// TIA Portal V17 export
// export: Created 2025-03-13T10:29:45.3472643Z, ExportSetting WithDefaults, DisplayName Totally Integrated Automation Portal, DisplayVersion V17 Update 8, DisplayName TIA Portal Openness, DisplayVersion V17 Update 8, DisplayName TIA Portal Version Control Interface, DisplayVersion V17, DisplayName SINAMICS Startdrive Advanced, DisplayVersion V17 SP2, DisplayName SINAMICS Startdrive G110M, G120, G120C, G120D, G120P, G115D, DisplayVersion V17 SP2, DisplayName SINAMICS Startdrive G130, G150, S120, S150, SINAMICS MV, S210, DisplayVersion V17 SP2, DisplayName STEP 7 Professional, DisplayVersion V17 Update 8, DisplayName SINUMERIK ONE STEP 7 Toolbox, DisplayVersion V17 Update 12, DisplayName SINUMERIK 840D sl STEP 7 Toolbox, DisplayVersion V17 Update 12, DisplayName STEP 7 Safety, DisplayVersion V17 Update 6, DisplayName WinCC Advanced, DisplayVersion V17 Update 8
FUNCTION "FC4020_PART_PRESENT_CONTROL_U02_STA_1" : Void   // FC4020, LAD
{ S7_Optimized_Access := 'TRUE' }
VERSION : 0.1
// stored: AutoNumber false, IsIECCheckEnabled false, SetENOAutomatically false, UDAEnableTagReadback false
   VAR_TEMP
      SENSOR_VALUE_AUX : Real;
      DIV_AUX : Real;
      RESULT_AUX : Real;
      TOTAL_AUX : Real;
      SUP_LIM : Real;
      INF_LIM : Real;
   END_VAR
BEGIN

REGION Network 1: PART PRESENT INPUT
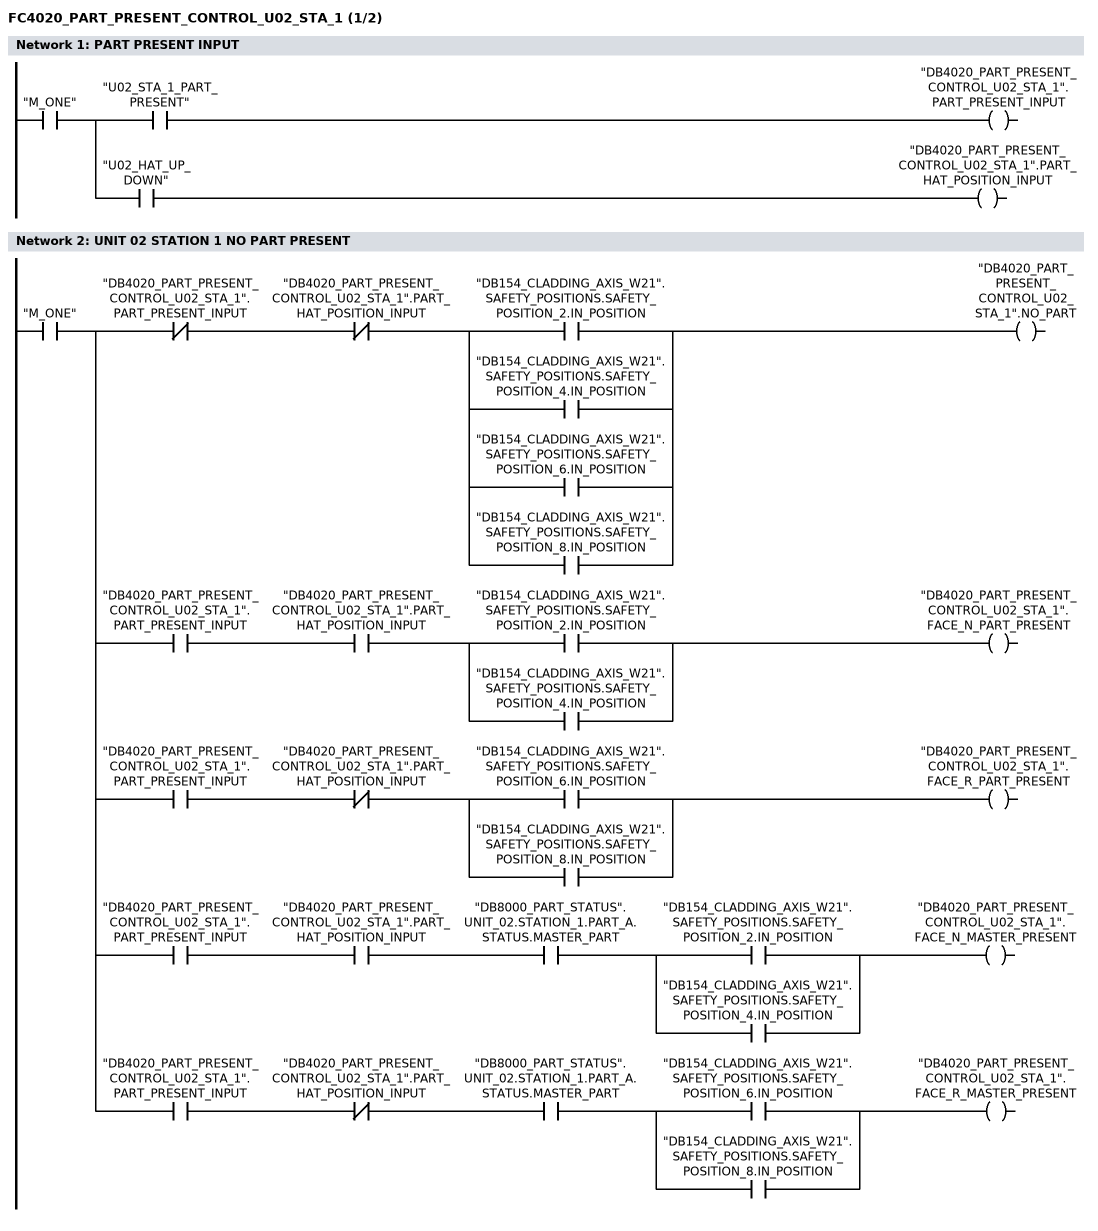
   RUNG wire#powerrail
      Contact( "M_ONE" )
      wire#w1
      Contact( "U02_STA_1_PART_PRESENT" )
      Coil( "DB4020_PART_PRESENT_CONTROL_U02_STA_1".PART_PRESENT_INPUT )
   END_RUNG
   RUNG wire#w1
      Contact( "U02_HAT_UP_DOWN" )
      Coil( "DB4020_PART_PRESENT_CONTROL_U02_STA_1".PART_HAT_POSITION_INPUT )
   END_RUNG
   // the same network as SCL:
   "DB4020_PART_PRESENT_CONTROL_U02_STA_1".PART_PRESENT_INPUT := "M_ONE" AND "U02_STA_1_PART_PRESENT";
   "DB4020_PART_PRESENT_CONTROL_U02_STA_1".PART_HAT_POSITION_INPUT := "M_ONE" AND "U02_HAT_UP_DOWN";
END_REGION

REGION Network 2: UNIT 02 STATION 1 NO PART PRESENT
   RUNG wire#powerrail
      Contact( "M_ONE" )
      wire#w1
      I_Contact( "DB4020_PART_PRESENT_CONTROL_U02_STA_1".PART_PRESENT_INPUT )
      I_Contact( "DB4020_PART_PRESENT_CONTROL_U02_STA_1".PART_HAT_POSITION_INPUT )
      wire#w2
      Contact( "DB154_CLADDING_AXIS_W21".SAFETY_POSITIONS.SAFETY_POSITION_2.IN_POSITION )
      wire#w3
      Coil( "DB4020_PART_PRESENT_CONTROL_U02_STA_1".NO_PART )
   END_RUNG
   RUNG wire#w2
      Contact( "DB154_CLADDING_AXIS_W21".SAFETY_POSITIONS.SAFETY_POSITION_4.IN_POSITION )
   END_RUNG wire#w3
   RUNG wire#w2
      Contact( "DB154_CLADDING_AXIS_W21".SAFETY_POSITIONS.SAFETY_POSITION_6.IN_POSITION )
   END_RUNG wire#w3
   RUNG wire#w2
      Contact( "DB154_CLADDING_AXIS_W21".SAFETY_POSITIONS.SAFETY_POSITION_8.IN_POSITION )
   END_RUNG wire#w3
   RUNG wire#w1
      Contact( "DB4020_PART_PRESENT_CONTROL_U02_STA_1".PART_PRESENT_INPUT )
      Contact( "DB4020_PART_PRESENT_CONTROL_U02_STA_1".PART_HAT_POSITION_INPUT )
      wire#w4
      Contact( "DB154_CLADDING_AXIS_W21".SAFETY_POSITIONS.SAFETY_POSITION_2.IN_POSITION )
      wire#w5
      Coil( "DB4020_PART_PRESENT_CONTROL_U02_STA_1".FACE_N_PART_PRESENT )
   END_RUNG
   RUNG wire#w4
      Contact( "DB154_CLADDING_AXIS_W21".SAFETY_POSITIONS.SAFETY_POSITION_4.IN_POSITION )
   END_RUNG wire#w5
   RUNG wire#w1
      Contact( "DB4020_PART_PRESENT_CONTROL_U02_STA_1".PART_PRESENT_INPUT )
      I_Contact( "DB4020_PART_PRESENT_CONTROL_U02_STA_1".PART_HAT_POSITION_INPUT )
      wire#w6
      Contact( "DB154_CLADDING_AXIS_W21".SAFETY_POSITIONS.SAFETY_POSITION_6.IN_POSITION )
      wire#w7
      Coil( "DB4020_PART_PRESENT_CONTROL_U02_STA_1".FACE_R_PART_PRESENT )
   END_RUNG
   RUNG wire#w6
      Contact( "DB154_CLADDING_AXIS_W21".SAFETY_POSITIONS.SAFETY_POSITION_8.IN_POSITION )
   END_RUNG wire#w7
   RUNG wire#w1
      Contact( "DB4020_PART_PRESENT_CONTROL_U02_STA_1".PART_PRESENT_INPUT )
      Contact( "DB4020_PART_PRESENT_CONTROL_U02_STA_1".PART_HAT_POSITION_INPUT )
      Contact( "DB8000_PART_STATUS".UNIT_02.STATION_1.PART_A.STATUS.MASTER_PART )
      wire#w8
      Contact( "DB154_CLADDING_AXIS_W21".SAFETY_POSITIONS.SAFETY_POSITION_2.IN_POSITION )
      wire#w9
      Coil( "DB4020_PART_PRESENT_CONTROL_U02_STA_1".FACE_N_MASTER_PRESENT )
   END_RUNG
   RUNG wire#w8
      Contact( "DB154_CLADDING_AXIS_W21".SAFETY_POSITIONS.SAFETY_POSITION_4.IN_POSITION )
   END_RUNG wire#w9
   RUNG wire#w1
      Contact( "DB4020_PART_PRESENT_CONTROL_U02_STA_1".PART_PRESENT_INPUT )
      I_Contact( "DB4020_PART_PRESENT_CONTROL_U02_STA_1".PART_HAT_POSITION_INPUT )
      Contact( "DB8000_PART_STATUS".UNIT_02.STATION_1.PART_A.STATUS.MASTER_PART )
      wire#w10
      Contact( "DB154_CLADDING_AXIS_W21".SAFETY_POSITIONS.SAFETY_POSITION_6.IN_POSITION )
      wire#w11
      Coil( "DB4020_PART_PRESENT_CONTROL_U02_STA_1".FACE_R_MASTER_PRESENT )
   END_RUNG
   RUNG wire#w10
      Contact( "DB154_CLADDING_AXIS_W21".SAFETY_POSITIONS.SAFETY_POSITION_8.IN_POSITION )
   END_RUNG wire#w11
   // the same network as SCL:
   "DB4020_PART_PRESENT_CONTROL_U02_STA_1".NO_PART := "M_ONE" AND NOT "DB4020_PART_PRESENT_CONTROL_U02_STA_1".PART_PRESENT_INPUT AND NOT "DB4020_PART_PRESENT_CONTROL_U02_STA_1".PART_HAT_POSITION_INPUT AND ("DB154_CLADDING_AXIS_W21".SAFETY_POSITIONS.SAFETY_POSITION_2.IN_POSITION OR "DB154_CLADDING_AXIS_W21".SAFETY_POSITIONS.SAFETY_POSITION_4.IN_POSITION OR "DB154_CLADDING_AXIS_W21".SAFETY_POSITIONS.SAFETY_POSITION_6.IN_POSITION OR "DB154_CLADDING_AXIS_W21".SAFETY_POSITIONS.SAFETY_POSITION_8.IN_POSITION);
   "DB4020_PART_PRESENT_CONTROL_U02_STA_1".FACE_N_PART_PRESENT := "M_ONE" AND "DB4020_PART_PRESENT_CONTROL_U02_STA_1".PART_PRESENT_INPUT AND "DB4020_PART_PRESENT_CONTROL_U02_STA_1".PART_HAT_POSITION_INPUT AND ("DB154_CLADDING_AXIS_W21".SAFETY_POSITIONS.SAFETY_POSITION_2.IN_POSITION OR "DB154_CLADDING_AXIS_W21".SAFETY_POSITIONS.SAFETY_POSITION_4.IN_POSITION);
   "DB4020_PART_PRESENT_CONTROL_U02_STA_1".FACE_R_PART_PRESENT := "M_ONE" AND "DB4020_PART_PRESENT_CONTROL_U02_STA_1".PART_PRESENT_INPUT AND NOT "DB4020_PART_PRESENT_CONTROL_U02_STA_1".PART_HAT_POSITION_INPUT AND ("DB154_CLADDING_AXIS_W21".SAFETY_POSITIONS.SAFETY_POSITION_6.IN_POSITION OR "DB154_CLADDING_AXIS_W21".SAFETY_POSITIONS.SAFETY_POSITION_8.IN_POSITION);
   "DB4020_PART_PRESENT_CONTROL_U02_STA_1".FACE_N_MASTER_PRESENT := "M_ONE" AND "DB4020_PART_PRESENT_CONTROL_U02_STA_1".PART_PRESENT_INPUT AND "DB4020_PART_PRESENT_CONTROL_U02_STA_1".PART_HAT_POSITION_INPUT AND "DB8000_PART_STATUS".UNIT_02.STATION_1.PART_A.STATUS.MASTER_PART AND ("DB154_CLADDING_AXIS_W21".SAFETY_POSITIONS.SAFETY_POSITION_2.IN_POSITION OR "DB154_CLADDING_AXIS_W21".SAFETY_POSITIONS.SAFETY_POSITION_4.IN_POSITION);
   "DB4020_PART_PRESENT_CONTROL_U02_STA_1".FACE_R_MASTER_PRESENT := "M_ONE" AND "DB4020_PART_PRESENT_CONTROL_U02_STA_1".PART_PRESENT_INPUT AND NOT "DB4020_PART_PRESENT_CONTROL_U02_STA_1".PART_HAT_POSITION_INPUT AND "DB8000_PART_STATUS".UNIT_02.STATION_1.PART_A.STATUS.MASTER_PART AND ("DB154_CLADDING_AXIS_W21".SAFETY_POSITIONS.SAFETY_POSITION_6.IN_POSITION OR "DB154_CLADDING_AXIS_W21".SAFETY_POSITIONS.SAFETY_POSITION_8.IN_POSITION);
END_REGION

REGION Network 3: UNIT 01 CLAMPED ANY PART
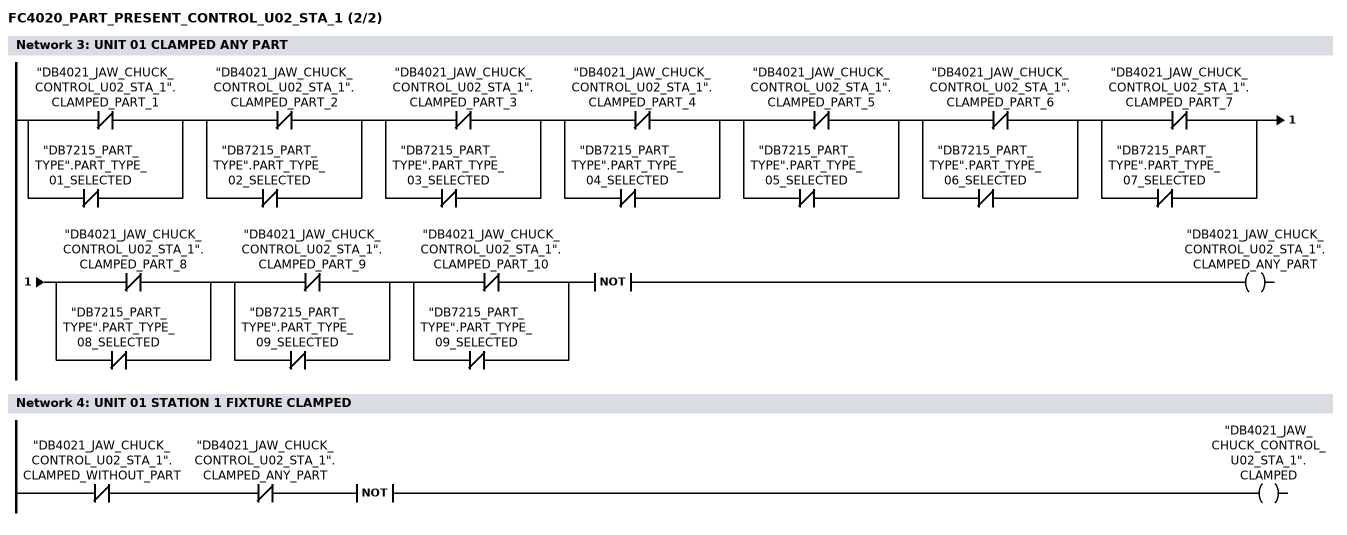
   RUNG wire#powerrail
      I_Contact( "DB4021_JAW_CHUCK_CONTROL_U02_STA_1".CLAMPED_PART_1 )
      wire#w1
      I_Contact( "DB4021_JAW_CHUCK_CONTROL_U02_STA_1".CLAMPED_PART_2 )
      wire#w2
      I_Contact( "DB4021_JAW_CHUCK_CONTROL_U02_STA_1".CLAMPED_PART_3 )
      wire#w3
      I_Contact( "DB4021_JAW_CHUCK_CONTROL_U02_STA_1".CLAMPED_PART_4 )
      wire#w4
      I_Contact( "DB4021_JAW_CHUCK_CONTROL_U02_STA_1".CLAMPED_PART_5 )
      wire#w5
      I_Contact( "DB4021_JAW_CHUCK_CONTROL_U02_STA_1".CLAMPED_PART_6 )
      wire#w6
      I_Contact( "DB4021_JAW_CHUCK_CONTROL_U02_STA_1".CLAMPED_PART_7 )
      wire#w7
      I_Contact( "DB4021_JAW_CHUCK_CONTROL_U02_STA_1".CLAMPED_PART_8 )
      wire#w8
      I_Contact( "DB4021_JAW_CHUCK_CONTROL_U02_STA_1".CLAMPED_PART_9 )
      wire#w9
      I_Contact( "DB4021_JAW_CHUCK_CONTROL_U02_STA_1".CLAMPED_PART_10 )
      wire#w10
      Not()
      Coil( "DB4021_JAW_CHUCK_CONTROL_U02_STA_1".CLAMPED_ANY_PART )
   END_RUNG
   RUNG wire#powerrail
      I_Contact( "DB7215_PART_TYPE".PART_TYPE_01_SELECTED )
   END_RUNG wire#w1
   RUNG wire#w1
      I_Contact( "DB7215_PART_TYPE".PART_TYPE_02_SELECTED )
   END_RUNG wire#w2
   RUNG wire#w2
      I_Contact( "DB7215_PART_TYPE".PART_TYPE_03_SELECTED )
   END_RUNG wire#w3
   RUNG wire#w3
      I_Contact( "DB7215_PART_TYPE".PART_TYPE_04_SELECTED )
   END_RUNG wire#w4
   RUNG wire#w4
      I_Contact( "DB7215_PART_TYPE".PART_TYPE_05_SELECTED )
   END_RUNG wire#w5
   RUNG wire#w5
      I_Contact( "DB7215_PART_TYPE".PART_TYPE_06_SELECTED )
   END_RUNG wire#w6
   RUNG wire#w6
      I_Contact( "DB7215_PART_TYPE".PART_TYPE_07_SELECTED )
   END_RUNG wire#w7
   RUNG wire#w7
      I_Contact( "DB7215_PART_TYPE".PART_TYPE_08_SELECTED )
   END_RUNG wire#w8
   RUNG wire#w8
      I_Contact( "DB7215_PART_TYPE".PART_TYPE_09_SELECTED )
   END_RUNG wire#w9
   RUNG wire#w9
      I_Contact( "DB7215_PART_TYPE".PART_TYPE_09_SELECTED )
   END_RUNG wire#w10
   // the same network as SCL:
   "DB4021_JAW_CHUCK_CONTROL_U02_STA_1".CLAMPED_ANY_PART := NOT ((NOT "DB4021_JAW_CHUCK_CONTROL_U02_STA_1".CLAMPED_PART_1 OR NOT "DB7215_PART_TYPE".PART_TYPE_01_SELECTED) AND (NOT "DB4021_JAW_CHUCK_CONTROL_U02_STA_1".CLAMPED_PART_2 OR NOT "DB7215_PART_TYPE".PART_TYPE_02_SELECTED) AND (NOT "DB4021_JAW_CHUCK_CONTROL_U02_STA_1".CLAMPED_PART_3 OR NOT "DB7215_PART_TYPE".PART_TYPE_03_SELECTED) AND (NOT "DB4021_JAW_CHUCK_CONTROL_U02_STA_1".CLAMPED_PART_4 OR NOT "DB7215_PART_TYPE".PART_TYPE_04_SELECTED) AND (NOT "DB4021_JAW_CHUCK_CONTROL_U02_STA_1".CLAMPED_PART_5 OR NOT "DB7215_PART_TYPE".PART_TYPE_05_SELECTED) AND (NOT "DB4021_JAW_CHUCK_CONTROL_U02_STA_1".CLAMPED_PART_6 OR NOT "DB7215_PART_TYPE".PART_TYPE_06_SELECTED) AND (NOT "DB4021_JAW_CHUCK_CONTROL_U02_STA_1".CLAMPED_PART_7 OR NOT "DB7215_PART_TYPE".PART_TYPE_07_SELECTED) AND (NOT "DB4021_JAW_CHUCK_CONTROL_U02_STA_1".CLAMPED_PART_8 OR NOT "DB7215_PART_TYPE".PART_TYPE_08_SELECTED) AND (NOT "DB4021_JAW_CHUCK_CONTROL_U02_STA_1".CLAMPED_PART_9 OR NOT "DB7215_PART_TYPE".PART_TYPE_09_SELECTED) AND (NOT "DB4021_JAW_CHUCK_CONTROL_U02_STA_1".CLAMPED_PART_10 OR NOT "DB7215_PART_TYPE".PART_TYPE_09_SELECTED));
END_REGION

REGION Network 4: UNIT 01 STATION 1 FIXTURE CLAMPED
   RUNG wire#powerrail
      I_Contact( "DB4021_JAW_CHUCK_CONTROL_U02_STA_1".CLAMPED_WITHOUT_PART )
      I_Contact( "DB4021_JAW_CHUCK_CONTROL_U02_STA_1".CLAMPED_ANY_PART )
      Not()
      Coil( "DB4021_JAW_CHUCK_CONTROL_U02_STA_1".CLAMPED )
   END_RUNG
   // the same network as SCL:
   "DB4021_JAW_CHUCK_CONTROL_U02_STA_1".CLAMPED := NOT (NOT "DB4021_JAW_CHUCK_CONTROL_U02_STA_1".CLAMPED_WITHOUT_PART AND NOT "DB4021_JAW_CHUCK_CONTROL_U02_STA_1".CLAMPED_ANY_PART);
END_REGION
END_FUNCTION
